(* CODESYS project Untitled1.project

Project tree, tasks and I/O mapping:
  Device : CODESYS Control Win V3, 3S - Smart Software Solutions GmbH, order no. 305021, version 3.5.11.30
    application Application
      libraries: Standard, * (System)
      task MainTask (cyclic, interval t#20ms, priority 1) calls PLC_PRG
      program PLC_PRG [SFC]: P1_active, P7_active, P2_active, P3_active, P4_active, P5_active, P6_active, Pcopo_active
*)

// Device/Application/PLC_PRG
PROGRAM PLC_PRG
VAR
	BT_LIGA: BOOL;
	PREPARAR: BOOL;
	SC: BOOL; //SENSOR DO COPO
	AL: BOOL; //ALIMENTADOR DE COPOS
	BT_A1: BOOL;
	BT_A2: BOOL;
	BT_A3: BOOL;
	BT_B1: BOOL;
	BT_B2: BOOL;
	BT_B3: BOOL;
	AUXAC: TIME; //TEMPO DO AÇUCAR
	AUXAG: TIME; //TEMPO DA AGUA
	AUXL: TIME; //TEMPO DA LEITE
	AUXCA: TIME; //TEMPO DA CAFE
	AUXCH: TIME; //TEMPO DO CHOCOLATE
	VR1: BOOL;
	VR2: BOOL;
	VR3: BOOL;
	VR4: BOOL;
	VR5: BOOL;
	L1: BOOL; //LAMPADA PREPARANDO
	L2: BOOL; //LAMPADA FALHA
END_VAR

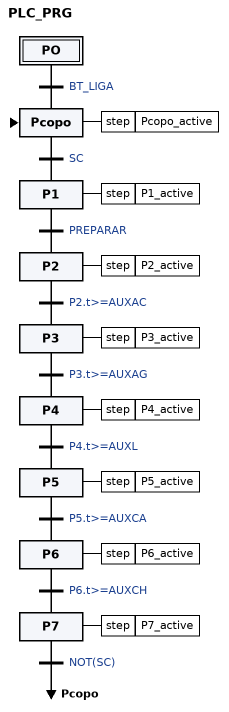
INITIAL_STEP PO:
END_STEP
TRANSITION FROM PO TO Pcopo
    := BT_LIGA;
END_TRANSITION
STEP Pcopo:
    Pcopo_active(N);  // step action
END_STEP
TRANSITION FROM Pcopo TO P1
    := SC;
END_TRANSITION
STEP P1:
    P1_active(N);  // step action
END_STEP
TRANSITION FROM P1 TO P2
    := PREPARAR;
END_TRANSITION
STEP P2:
    P2_active(N);  // step action
END_STEP
TRANSITION FROM P2 TO P3
    := P2.t>=AUXAC;
END_TRANSITION
STEP P3:
    P3_active(N);  // step action
END_STEP
TRANSITION FROM P3 TO P4
    := P3.t>=AUXAG;
END_TRANSITION
STEP P4:
    P4_active(N);  // step action
END_STEP
TRANSITION FROM P4 TO P5
    := P4.t>=AUXL;
END_TRANSITION
STEP P5:
    P5_active(N);  // step action
END_STEP
TRANSITION FROM P5 TO P6
    := P5.t>=AUXCA;
END_TRANSITION
STEP P6:
    P6_active(N);  // step action
END_STEP
TRANSITION FROM P6 TO P7
    := P6.t>=AUXCH;
END_TRANSITION
STEP P7:
    P7_active(N);  // step action
END_STEP
TRANSITION FROM P7 TO Pcopo
    := NOT(SC);
END_TRANSITION

ACTION P1_active:
L2:=FALSE;
//SELEÇÃO DO TEMPO DO AÇÚCAR
IF BT_A1 AND NOT(BT_A2) AND NOT (BT_A3) THEN 
	AUXAC:=T#0S;
END_IF

IF BT_A2 AND NOT(BT_A1) AND NOT (BT_A3) THEN 
	AUXAC:=T#3S;
END_IF

IF BT_A3 AND NOT(BT_A1) AND NOT (BT_A2) THEN 
	AUXAC:=T#6S;
END_IF

//SELEÇÃO DOS TEMPOS DAS BEBIDA
IF BT_B1 AND NOT (BT_B2) AND NOT (BT_B3) THEN 
	AUXCA:=T#3S;
	AUXAG:=T#5S;
END_IF

IF BT_B2 AND NOT (BT_B1) AND NOT (BT_B3) THEN 
	AUXCA:=T#2S;
	AUXL:=T#3S;
	AUXAG:=T#7S;
END_IF

IF BT_B3 AND NOT (BT_B1) AND NOT (BT_B2) THEN 
	AUXCH:=T#3S;
	AUXL:=T#2S;
	AUXAG:=T#7S;
END_IF
END_ACTION

ACTION P7_active:
//ZERANDO TIMES
AUXAC:= T#0S;
AUXAG:= T#0S;
AUXL:= T#0S;
AUXCA:= T#0S;
AUXCH:= T#0S;

VR1:=FALSE;
VR2:=FALSE;
VR3:=FALSE;
VR4:=FALSE;
VR5:=FALSE;

L1:= FALSE;
END_ACTION

ACTION P2_active:

VR1:=FALSE;
VR2:=FALSE;
VR3:=FALSE;
VR4:=TRUE;
VR5:=FALSE;
L1:= TRUE;
AL:= FALSE;
END_ACTION

ACTION P3_active:

VR1:=FALSE;
VR2:=FALSE;
VR3:=FALSE;
VR4:=FALSE;
VR5:=TRUE;
END_ACTION

ACTION P4_active:

VR1:=FALSE;
VR2:=TRUE;
VR3:=FALSE;
VR4:=FALSE;
VR5:=FALSE;
END_ACTION

ACTION P5_active:
VR1:=TRUE;
VR2:=FALSE;
VR3:=FALSE;
VR4:=FALSE;
VR5:=FALSE;
END_ACTION

ACTION P6_active:
VR1:=FALSE;
VR2:=FALSE;
VR3:=TRUE;
VR4:=FALSE;
VR5:=FALSE;
END_ACTION

ACTION Pcopo_active:
IF NOT(SC) THEN
	L2:=TRUE;
	AL:= TRUE;
	ELSE
	AL:= FALSE;
	L2:=FALSE;
END_IF
END_ACTION

END_PROGRAM
